Staubli VAL3: onDefault.pgx

program onDefault()
begin
  aioSet(MbAO_bAxis7Home,0)
  aioSet(MbAO_bResetErr,0)

end
